{attribute 'pack_mode' := '1'} 
TYPE ST_Packed :
STRUCT
	bMember  		: BOOL;
    dtMember 		: DT;
	fMember   		: LREAL;
END_STRUCT
END_TYPE

(* stored: Version 1.1.0.1
   DUT ST_Packed: Id {e065de16-737d-4d99-829b-e9160723d009} *)
